Yaskawa INFORM job: FRONT_WELD_0ST-2_4040_V2.JBI

/JOB
//NAME FRONT_WELD_0ST-2_4040_V2
///FOLDERNAME 02-SKRZYNIE_JOBS
//POS
///NPOS 123,123,0,25,0,0
///TOOL 0
///POSTYPE PULSE
///PULSE
C00000=1212,-39190,49707,1936,-15809,-581
C00001=-55064,-17017,13106,20113,45767,-35735
C00002=-85641,-3161,12660,31281,67420,-55579
C00003=-77611,9747,38455,32702,57795,-55547
C00004=-77611,9747,38455,32702,57795,-55547
C00005=-80481,23547,61641,37204,60115,-56891
C00006=-80479,11681,28780,33754,71138,-52780
C00007=-72933,30277,53605,31576,73074,-55586
C00008=-73419,29451,52323,31530,73467,-55649
C00009=-73173,32098,57907,31817,71820,-56064
C00010=-72991,37471,72685,33001,66631,-57677
C00011=-82806,26311,53816,38180,73291,-53604
C00012=-71695,3747,16001,30713,64750,-51022
C00013=-70421,5575,20105,30867,63066,-51036
C00014=-35893,-19818,-4542,23004,50197,-40345
C00015=-37830,-23193,-8618,23571,50957,-40982
C00016=11136,-28839,-12562,1025,41780,-20887
C00017=20436,-26886,-6789,-12590,38175,-10721
C00018=58488,-10629,5191,-26833,51354,2977
C00019=55110,-17412,-5825,-19778,50988,-2825
C00020=79390,11759,28162,-35512,71262,52960
C00021=82927,23281,58968,-48274,65531,63493
C00022=83399,22743,58163,-48180,65853,63532
C00023=83221,24593,61395,-48465,65231,63817
C00024=82927,34411,85507,-52086,59386,67513
C00025=83936,23300,58997,-48174,66010,63700
C00026=83936,23300,58997,-48174,66010,63700
C00027=76815,18630,46530,-37158,64288,54543
C00028=79390,11759,28162,-35512,71262,52960
C00029=10831,-54278,-29128,-6468,39852,-5090
C00030=-67200,-10549,24402,-3189,24913,-39001
C00031=-75122,-2194,12822,3152,39225,-43427
C00032=-77516,10189,32861,8493,33365,-45533
C00033=-75154,17675,49539,7913,27349,-44943
C00034=-68113,10120,39417,1165,28259,-40458
C00035=-67114,5383,31515,9208,32648,-43213
C00036=-66450,3998,29285,10896,33890,-43630
C00037=-66374,3101,28136,14657,35566,-44954
C00038=-66747,-26,23691,26916,43760,-49061
C00039=-70537,4638,30761,35492,50867,-52773
C00040=-77050,-3138,8526,33226,61087,-51698
C00041=-67200,-10549,24402,-3189,24913,-39001
C00042=0,-52280,40443,83103,28146,-16510
C00043=99993,-20782,22705,-13349,24734,56519
C00044=67200,-10549,24402,3189,24913,39001
C00045=75122,-2194,12822,-3152,39225,43427
C00046=74323,5203,27259,-5972,33194,43789
C00047=74015,16414,48063,-6821,27325,44224
C00048=56519,1138,28747,9235,29393,33453
C00049=55467,619,28251,10155,29461,32830
C00050=56374,-724,25854,4078,30541,35419
C00051=56321,-6570,17381,-17816,37906,43384
C00052=68252,956,25699,-34035,49810,51639
C00053=77050,-3138,8526,-33226,61087,51698
C00054=67200,-10549,24402,3189,24913,39001
C00055=0,-52280,40443,-83103,28146,16510
C00056=-99993,-20782,22705,13349,24734,-56519
C00057=-91125,453,39555,30378,52425,-51131
C00058=-81425,-5449,14825,37552,56592,-47667
C00059=-81425,-10835,-2515,34915,62871,-45127
C00060=-79239,4305,16082,37593,68846,-50182
C00061=-83523,16585,41906,47112,68321,-58375
C00062=-83466,26209,67230,50527,61769,-62335
C00063=-83442,29914,76031,51903,59779,-63702
C00064=-84288,15645,43522,43516,65950,-57098
C00065=-90096,4679,14083,37467,76581,-51973
C00066=-87885,29238,52923,40761,81198,69685
C00067=-84355,23847,39024,40698,83720,72224
C00068=-82166,27958,47897,41071,80495,71788
C00069=-78317,33303,56220,41538,77506,72130
C00070=-90480,18737,31939,47254,81986,71631
C00071=-94217,10634,17426,46901,86469,-59967
C00072=-81425,-10835,-2515,34915,62871,-45127
C00073=-81425,-5449,14825,37552,56592,-47667
C00074=-94290,-610,44819,32366,49686,-53459
C00075=0,-55136,17047,60468,32096,-4233
C00076=99993,-20782,22705,-13349,24734,56519
C00077=91125,453,39555,-30378,52425,51131
C00078=81425,-5449,14825,-37552,56592,47667
C00079=81425,-10835,-2515,-34915,62871,45127
C00080=79239,4305,16082,-37593,68846,50182
C00081=80765,23031,47100,-43000,73595,58456
C00082=80765,35859,79857,-46269,64609,63023
C00083=81236,37975,84040,-46627,63953,63603
C00084=79256,17348,34699,-33448,76412,88212
C00085=79932,23608,50901,-39863,71219,88955
C00086=76220,30771,63034,-41386,67395,88927
C00087=86322,16060,37848,-39554,76452,89287
C00088=87424,-1569,9538,-38190,72401,52253
C00089=81425,-10835,-2515,-34915,62871,45127
C00090=92850,-11266,9233,-39092,60986,50964
C00091=28366,-40369,19479,-5635,23506,17663
C00092=-80334,-19501,31260,21216,42469,-40219
C00093=-80621,-32280,-9061,25825,59412,-41877
C00094=-80621,-37319,-22868,24573,64555,-40576
C00095=-75108,-2453,16462,35304,60348,-42510
C00096=-72509,6961,33136,36537,55809,-43202
C00097=-35516,-19804,6201,28214,41034,-31537
C00098=-39606,-22901,-1163,28356,44724,-32188
C00099=15344,-29112,-5358,-2858,33820,-6852
C00100=13899,-24312,2834,-1929,31756,-7563
C00101=57847,-8649,16006,-27199,42364,12903
C00102=60973,-17187,4937,-27817,44388,13718
C00103=60973,-17187,4937,-27817,44388,13718
C00104=-13287,-42463,-12044,19170,31021,-23010
C00105=-17374,-21287,20534,22794,29118,-26096
C00106=13276,-20759,18622,-1911,29377,-7028
C00107=18345,-20450,18118,-4901,30133,-4565
C00108=40008,-14355,19238,-14842,35994,4442
C00109=41528,-14133,18797,-15449,36702,5040
C00110=57001,-5890,26499,-21893,40771,11494
C00111=64054,-19541,3059,-29141,44956,15011
C00112=51466,-33957,-1499,-46586,51805,23434
C00113=17032,-20770,22044,-28854,30468,11088
C00114=-10379,-19290,13742,-8195,38792,-5467
C00115=-15395,-18849,14560,-5818,37558,-7698
C00116=-40849,-13899,18629,9604,35747,-20285
C00117=-41848,-12775,19702,10127,35967,-20750
C00118=-57173,-4328,27598,17453,39247,-27560
C00119=-71680,-19835,10874,33863,39440,-36917
C00120=-20806,-37586,-12792,9951,42782,-18031
///LIMIT ON
C00121=29087,-45372,27330,-13325,19529,9021
C00122=0,-35121,73515,0,-2982,0
///LIMIT OFF
BC00000=678863
BC00001=730815
BC00002=734074
BC00003=734074
BC00004=734074
BC00005=734074
BC00006=750936
BC00007=750938
BC00008=750938
BC00009=750938
BC00010=750938
BC00011=750938
BC00012=750938
BC00013=750938
BC00014=750938
BC00015=750938
BC00016=750938
BC00017=750937
BC00018=750938
BC00019=750939
BC00020=750939
BC00021=750937
BC00022=750937
BC00023=750937
BC00024=750937
BC00025=750937
BC00026=750937
BC00027=750939
BC00028=750939
BC00029=746449
BC00030=722597
BC00031=751774
BC00032=751777
BC00033=751777
BC00034=751774
BC00035=751775
BC00036=751776
BC00037=751776
BC00038=751777
BC00039=751777
BC00040=751777
BC00041=722597
BC00042=651203
BC00043=651203
BC00044=722597
BC00045=751774
BC00046=751777
BC00047=751777
BC00048=751777
BC00049=751777
BC00050=751782
BC00051=751789
BC00052=751778
BC00053=751777
BC00054=722597
BC00055=651203
BC00056=651203
BC00057=688665
BC00058=734468
BC00059=753865
BC00060=753867
BC00061=753867
BC00062=753867
BC00063=753867
BC00064=753867
BC00065=754443
BC00066=753867
BC00067=767806
BC00068=767806
BC00069=767806
BC00070=767806
BC00071=767806
BC00072=753865
BC00073=734468
BC00074=688665
BC00075=688951
BC00076=651203
BC00077=688665
BC00078=734468
BC00079=753865
BC00080=753867
BC00081=753867
BC00082=753867
BC00083=753867
BC00084=753867
BC00085=753867
BC00086=753867
BC00087=753867
BC00088=753867
BC00089=753865
BC00090=734468
BC00091=665480
BC00092=679958
BC00093=699518
BC00094=737823
BC00095=737823
BC00096=737823
BC00097=737821
BC00098=737823
BC00099=737823
BC00100=737823
BC00101=737821
BC00102=737823
BC00103=730488
BC00104=737823
BC00105=737823
BC00106=737819
BC00107=737819
BC00108=737821
BC00109=737865
BC00110=737821
BC00111=737823
BC00112=737823
BC00113=737819
BC00114=737821
BC00115=737821
BC00116=737823
BC00117=737823
BC00118=737823
BC00119=737823
BC00120=734415
BC00121=621191
BC00122=513349
///POSTYPE BASE
///RECTAN
///RCONF 0,0,0,0,0,0,0,0,0,0,0,0,0,0,0,0,0,0,0,0,0,0,0,0
P00021=6.550,-0.003,-5.735,0.0000,0.0000,0.0000
P00022=5.943,-0.018,-6.388,0.0000,0.0000,0.0000
P00023=7.025,-0.019,-7.168,0.0000,0.0000,0.0000
P00024=5.926,-0.047,-4.777,0.0000,0.0000,0.0000
P00350=11.519,-0.008,1.149,0.0000,0.0000,0.0000
P00351=13.563,-0.027,-0.653,0.0000,0.0000,0.0000
P00352=13.252,-0.027,-0.827,0.0000,0.0000,0.0000
P00353=10.971,-0.082,0.776,0.0000,0.0000,0.0000
P00399=-2.449,0.031,8.825,0.0000,0.0000,0.0000
P00400=5.920,-3.503,-0.024,0.0000,0.0000,0.0000
P00401=3.430,-0.021,1.131,0.0000,0.0000,0.0000
P00402=-0.253,1.107,3.062,0.0000,0.0000,0.0000
P00403=-3.666,-0.015,5.328,0.0000,0.0000,0.0000
P00405=2.420,0.007,1.427,0.0000,0.0000,0.0000
P00406=3.513,-0.022,0.429,0.0000,0.0000,0.0000
P00415=-1.781,-1.303,3.250,0.0000,0.0000,0.0000
P00416=0.027,1.119,3.078,0.0000,0.0000,0.0000
P00420=-0.017,0.555,2.209,0.0000,0.0000,0.0000
P00421=4.378,0.044,2.315,0.0000,0.0000,0.0000
P00422=2.474,0.026,-1.450,0.0000,0.0000,0.0000
P00423=4.044,0.004,-2.619,0.0000,0.0000,0.0000
P00424=-0.387,-0.003,1.304,0.0000,0.0000,0.0000
P00425=-1.050,0.029,1.708,0.0000,0.0000,0.0000
P00426=0.002,-0.749,-0.024,0.0000,0.0000,0.0000
P00427=-1.030,-0.025,3.232,0.0000,0.0000,0.0000
//INST
///DATE 2025/03/28 08:40
///ATTR SC,RW
///GROUP1 RB1,BS1
NOP
'**********************
'**********************
'POCZATEK SPAWANIA PRZOD
'**********************
'**********************
MOVJ C00000 BC00000 VJ=60.00
MOVL C00001 BC00001 V=416.7
MOVJ C00002 BC00002 VJ=10.00
MOVJ C00003 BC00003 VJ=10.00
MOVL C00004 BC00004 V=150.0
MOVL C00005 BC00005 V=150.0
'**********************
'W41A SIDE
'**********************
MOVL C00006 BC00006 V=250.0
SFTON P0402
MOVL C00007 BC00007 V=66.7 PL=0
REFP 1 C00008 BC00008
REFP 2 C00009 BC00009
MACRO1 MJ#(0) ARGF14
ARCON
WVON WEV#(5)
MOVL C00010 BC00010 V=9.2
ARCOF
WVOF
SFTOF
MOVL C00011 BC00011 V=166.7
'**********************
'W41A FRONT
'**********************
MOVL C00012 BC00012 V=250.0
SFTON P0350
MOVL C00013 BC00013 V=66.7 PL=0
SFTOF
MACRO1 MJ#(0) ARGF21
ARCON
WVON WEV#(2)
SFTON P0351
MOVL C00014 BC00014 V=8.3
SFTOF
ARCOF
WVOF
MOVL C00015 BC00015 V=166.7
'**********************
'W41B FRONT
'**********************
MOVL C00016 BC00016 V=250.0
SFTON P0352
MOVL C00017 BC00017 V=66.7 PL=0
SFTOF
MACRO1 MJ#(0) ARGF21
ARCON
WVON WEV#(2)
SFTON P0353
MOVL C00018 BC00018 V=8.3
SFTOF
ARCOF
WVOF
MOVL C00019 BC00019 V=166.7
MOVL C00020 BC00020 V=100.0
'**********************
'W41A SIDE
'**********************
SFTON P0400
MOVL C00021 BC00021 V=66.7 PL=0
MACRO1 MJ#(0) ARGF21
REFP 1 C00022 BC00022
REFP 2 C00023 BC00023
ARCON
WVON WEV#(5)
MOVL C00024 BC00024 V=8.3
ARCOF
WVOF
SFTOF
MOVJ C00025 BC00025 VJ=10.00
MOVL C00026 BC00026 V=133.3
MOVL C00027 BC00027 V=166.7
MOVL C00028 BC00028 V=166.7
MOVL C00029 BC00029 V=333.3
MOVJ C00030 BC00030 VJ=20.00
MOVJ C00031 BC00031 VJ=20.00
'**********************
'W42A.1
'**********************
'POPRAWIC
MOVL C00032 BC00032 V=500.0
SFTON P0403
MOVL C00033 BC00033 V=66.7 PL=0
MACRO1 MJ#(0) ARGF9
ARCON
MOVL C00034 BC00034 V=9.2
SFTON P0416
MOVL C00035 BC00035 V=9.2
MOVL C00036 BC00036 V=9.2
MOVL C00037 BC00037 V=9.2
SFTON P0421
MOVL C00038 BC00038 V=9.2
SFTON P0402
MOVL C00039 BC00039 V=9.2
ARCOF
MOVL C00040 BC00040 V=500.0
SFTOF
MOVJ C00041 BC00041 VJ=15.00
'W42B.1
MOVJ C00042 BC00042 VJ=30.00
MOVJ C00043 BC00043 VJ=30.00
MOVJ C00044 BC00044 VJ=30.00
MOVJ C00045 BC00045 VJ=30.00
'**********************
'W42B.1
'**********************
MOVL C00046 BC00046 V=500.0
SFTON P0399
MOVL C00047 BC00047 V=166.7 PL=0
MACRO1 MJ#(0) ARGF9
ARCON
SFTON P0415
MOVL C00048 BC00048 V=9.2
MOVL C00049 BC00049 V=9.2
MOVL C00050 BC00050 V=9.2
SFTON P0427
MOVL C00051 BC00051 V=9.2
SFTON P0400
MOVL C00052 BC00052 V=9.2
ARCOF
MOVL C00053 BC00053 V=500.0
SFTOF
MOVJ C00054 BC00054 VJ=25.00
'W42A.2
MOVJ C00055 BC00055 VJ=40.00
MOVJ C00056 BC00056 VJ=30.00
MOVJ C00057 BC00057 VJ=30.00
MOVJ C00058 BC00058 VJ=30.00
MOVJ C00059 BC00059 VJ=30.00
'**********************
'W42A.2
'**********************
MOVL C00060 BC00060 V=500.0
SFTON P0420
MOVL C00061 BC00061 V=166.7 PL=0
SFTOF
MACRO1 MJ#(0) ARGF9
ARCON
WVON WEV#(6)
MOVL C00062 BC00062 V=9.2
SFTON P0402
MOVL C00063 BC00063 V=9.2
ARCOF
WVOF
MOVL C00064 BC00064 V=166.7
MOVJ C00065 BC00065 VJ=20.00
MOVJ C00066 BC00066 VJ=20.00
MOVL C00067 BC00067 V=250.0
MOVL C00068 BC00068 V=166.7
ARCON
MOVL C00069 BC00069 V=10.8
ARCOF
MOVL C00070 BC00070 V=166.7
MOVJ C00071 BC00071 VJ=20.00
SFTOF
MOVJ C00072 BC00072 VJ=30.00
MOVJ C00073 BC00073 VJ=30.00
MOVJ C00074 BC00074 VJ=30.00
'W42B.2
MOVJ C00075 BC00075 VJ=30.00
MOVJ C00076 BC00076 VJ=30.00
MOVJ C00077 BC00077 VJ=30.00
MOVJ C00078 BC00078 VJ=30.00
MOVJ C00079 BC00079 VJ=30.00
'**********************
'W42B.2
'**********************
MOVL C00080 BC00080 V=500.0
SFTON P0426
MOVL C00081 BC00081 V=166.7 PL=0
SFTOF
MACRO1 MJ#(0) ARGF9
ARCON
WVON WEV#(6)
MOVL C00082 BC00082 V=9.2
SFTON P0400
MOVL C00083 BC00083 V=9.2
ARCOF
WVOF
SFTOF
MOVJ C00084 BC00084 VJ=10.00
SFTON P0400
MOVL C00085 BC00085 V=166.7
ARCON
MOVL C00086 BC00086 V=10.8
ARCOF
MOVL C00087 BC00087 V=250.0
MOVL C00088 BC00088 V=500.0
SFTOF
MOVJ C00089 BC00089 VJ=20.00
MOVJ C00090 BC00090 VJ=30.00
'W42A.3
MOVJ C00091 BC00091 VJ=20.00
MOVJ C00092 BC00092 VJ=20.00
MOVJ C00093 BC00093 VJ=30.00
MOVJ C00094 BC00094 VJ=30.00
'**********************
'W42A.3
'**********************
MOVL C00095 BC00095 V=500.0
SFTON P0021
MOVL C00096 BC00096 V=166.7 PL=0
MACRO1 MJ#(0) ARGF9
ARCON
WVON WEV#(2)
SFTON P0022
MOVL C00097 BC00097 V=9.2
ARCOF
WVOF
MOVL C00098 BC00098 V=500.0
SFTOF
'**********************
'W42B.3
'**********************
MOVL C00099 BC00099 V=500.0
SFTON P0023
MOVL C00100 BC00100 V=166.7 PL=0
ARCON
WVON WEV#(2)
SFTON P0024
MOVL C00101 BC00101 V=9.2
ARCOF
WVOF
MOVL C00102 BC00102 V=500.0
SFTOF
MOVJ C00103 BC00103 VJ=20.00
'**********************
'GORA L
'**********************
MOVL C00104 BC00104 V=500.0
SFTON P0401
MOVL C00105 BC00105 V=166.7 PL=0
MACRO1 MJ#(0) ARGF9
ARCON
MOVL C00106 BC00106 V=11.7
SFTON P0424
MOVL C00107 BC00107 V=11.7
SFTON P0425
MOVL C00108 BC00108 V=11.7
SFTON P0406
MOVL C00109 BC00109 V=11.7
MOVL C00110 BC00110 V=11.7
ARCOF
MOVL C00111 BC00111 V=500.0
SFTOF
'**********************
'GORA P
'**********************
MOVL C00112 BC00112 V=166.7
SFTON P0401
MOVL C00113 BC00113 V=166.7 PL=0
ARCON
MOVL C00114 BC00114 V=11.7
SFTON P0423
MOVL C00115 BC00115 V=11.7
SFTON P0422
MOVL C00116 BC00116 V=11.7
SFTON P0405
MOVL C00117 BC00117 V=11.7
MOVL C00118 BC00118 V=11.7
ARCOF
MOVL C00119 BC00119 V=500.0
SFTOF
MOVJ C00120 BC00120 VJ=20.00
MOVJ C00121 BC00121 VJ=30.00
MOVJ C00122 BC00122 VJ=30.00
'KONIEC SPAWANIA FRONTU
END
